(* PLC project  *)

CONFIGURATION XB_EC_12
END_CONFIGURATION
